// TIA Portal V19 export
VAR_GLOBAL   // PLC tag table "Level_Tags"
   Pump1_Mode AT %M5.1 : Bool;   // Running Mode ( Auto or Manual)
   Pump1_Start_Manual AT %M5.2 : Bool;   // Start Manual Mode
   Pump1_Stop_Manual AT %M5.3 : Bool;   // Stop Manual Mode
   Pump1_Start_Auto AT %M5.4 : Bool;   // Start Auto Mode
   Pump1_Stop_Auto AT %M5.5 : Bool;   // Stop Auto Mode
   Level_High AT %M5.6 : Bool;   // High Level Reached
   Level_Low AT %M5.7 : Bool;   // Low Level Reached
   Timer_Setting_Run AT %MD6 : DInt;   // Timer Settings for Running
   Pump1_Overload AT %M10.0 : Bool;   // Pump Overloaded
   Pump1_Reset_Fault AT %M10.1 : Bool;   // Pump Reset Fault
   Pump1 AT %Q0.0 : Bool;   // Pump 1 - Output
   Pump1_Fault AT %M10.2 : Bool;   // Pump 1 Fault Status
   Pump1_Run_Auto_Activated AT %M10.3 : Bool;   // Pump 1 Running in Auto
   Level_Meter AT %MW12 : Int;   // Level Meter Reading
   Sensor_Real AT %QD2 : Real;   // Real Sensor Reading ( Tank Level)
   High_SP AT %MD14 : Real;   // High Setpoint
   Low_SP AT %MD18 : Real;   // Low Setpoint
END_VAR
